// TIA Portal V15.1 export
// export: Created 2024-06-21T08:41:24.8000598Z, ExportSetting WithDefaults, DisplayName Totally Integrated Automation Portal, DisplayVersion V15.1 Update 5, DisplayName TIA Portal Openness, DisplayVersion V15.1 Update 5, DisplayName SINAMICS Startdrive Advanced, DisplayVersion V15.1, DisplayName G130, G150, S120, S150, SINAMICS MV, S210, DisplayVersion V15.1, DisplayName G110M, G120, G120C, G120D, G120P, DisplayVersion V15.1, DisplayName STEP 7 Professional, DisplayVersion V15.1 Update 5, DisplayName STEP 7 Safety, DisplayVersion V15.1, DisplayName WinCC Professional, DisplayVersion V15.1 Update 5, DisplayName SIMATIC Visualization Architect, DisplayVersion V15.1
FUNCTION "209230ZM01DataHandling" : Void   // FC404, FBD
TITLE = 209230ZM01 Data Handling
{ S7_Optimized_Access := 'FALSE' }
AUTHOR : VCC
VERSION : 0.1
// stored: AutoNumber false, IsIECCheckEnabled false, SetENOAutomatically False, UDAEnableTagReadback false
   VAR_OUTPUT
      O_AlarmA : Bool;   // Alarm A
      O_AlarmB : Bool;   // Alarm B
      O_AlarmC : Bool;   // Alarm C
      O_AlarmD : Bool;   // Alarm D
      O_AlarmABCondition : Bool;   // Alarm AB Condition
      H_IAnim : Word;   // Icon Animation
   END_VAR
BEGIN

REGION Network 1: **** 4.6 - Machine status - Indications **** Icon animation
   // Icon animation
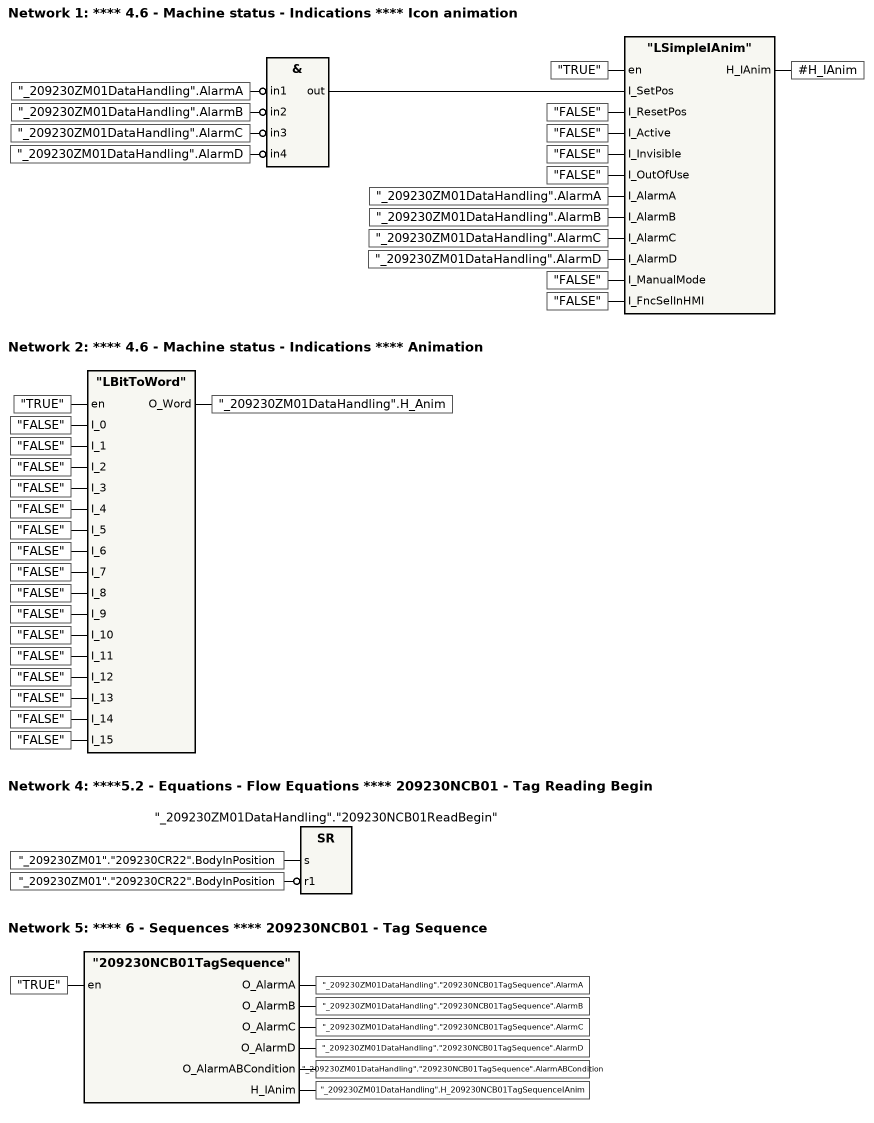
   IF "TRUE" THEN
       "LSimpleIAnim"(I_SetPos := NOT "_209230ZM01DataHandling".AlarmA AND NOT "_209230ZM01DataHandling".AlarmB AND NOT "_209230ZM01DataHandling".AlarmC AND NOT "_209230ZM01DataHandling".AlarmD,
                      I_ResetPos := "FALSE",
                      I_Active := "FALSE",
                      I_Invisible := "FALSE",
                      I_OutOfUse := "FALSE",
                      I_AlarmA := "_209230ZM01DataHandling".AlarmA,
                      I_AlarmB := "_209230ZM01DataHandling".AlarmB,
                      I_AlarmC := "_209230ZM01DataHandling".AlarmC,
                      I_AlarmD := "_209230ZM01DataHandling".AlarmD,
                      I_ManualMode := "FALSE",
                      I_FncSelInHMI := "FALSE",
                      H_IAnim => #H_IAnim);
   END_IF;
END_REGION

REGION Network 2: **** 4.6 - Machine status - Indications **** Animation
   // Animation
   IF "TRUE" THEN
       "LBitToWord"(I_0 := "FALSE",
                    I_1 := "FALSE",
                    I_2 := "FALSE",
                    I_3 := "FALSE",
                    I_4 := "FALSE",
                    I_5 := "FALSE",
                    I_6 := "FALSE",
                    I_7 := "FALSE",
                    I_8 := "FALSE",
                    I_9 := "FALSE",
                    I_10 := "FALSE",
                    I_11 := "FALSE",
                    I_12 := "FALSE",
                    I_13 := "FALSE",
                    I_14 := "FALSE",
                    I_15 := "FALSE",
                    O_Word => "_209230ZM01DataHandling".H_Anim);
   END_IF;
END_REGION

NETWORK
TITLE = **** 4.6 - Machine Status - Indications **** Animation DB number
// DB number
      OPN   "_209230ZM01DataHandling";
      L     DBNO;
      T     "_209230ZM01DataHandling".H_DBnr;

REGION Network 4: ****5.2 - Equations - Flow Equations **** 209230NCB01 - Tag Reading Begin
   // Singal to start the reading of the Tag
   IF "_209230ZM01"."209230CR22".BodyInPosition THEN
       "_209230ZM01DataHandling"."209230NCB01ReadBegin" := TRUE;   // SR flip-flop
   END_IF;
   IF NOT "_209230ZM01"."209230CR22".BodyInPosition THEN
       "_209230ZM01DataHandling"."209230NCB01ReadBegin" := FALSE;
   END_IF;
END_REGION

REGION Network 5: **** 6 - Sequences **** 209230NCB01 - Tag Sequence
   // Tag Sequence
   IF "TRUE" THEN
       "209230NCB01TagSequence"(O_AlarmA => "_209230ZM01DataHandling"."209230NCB01TagSequence".AlarmA,
                               O_AlarmB => "_209230ZM01DataHandling"."209230NCB01TagSequence".AlarmB,
                               O_AlarmC => "_209230ZM01DataHandling"."209230NCB01TagSequence".AlarmC,
                               O_AlarmD => "_209230ZM01DataHandling"."209230NCB01TagSequence".AlarmD,
                               O_AlarmABCondition => "_209230ZM01DataHandling"."209230NCB01TagSequence".AlarmABCondition,
                               H_IAnim => "_209230ZM01DataHandling".H_209230NCB01TagSequenceIAnim);
   END_IF;
END_REGION

REGION Network 6: **** 7.1 - Submodule - Non Machine **** 209230NCB01 - VIDS Master
   // VIDS Master Module
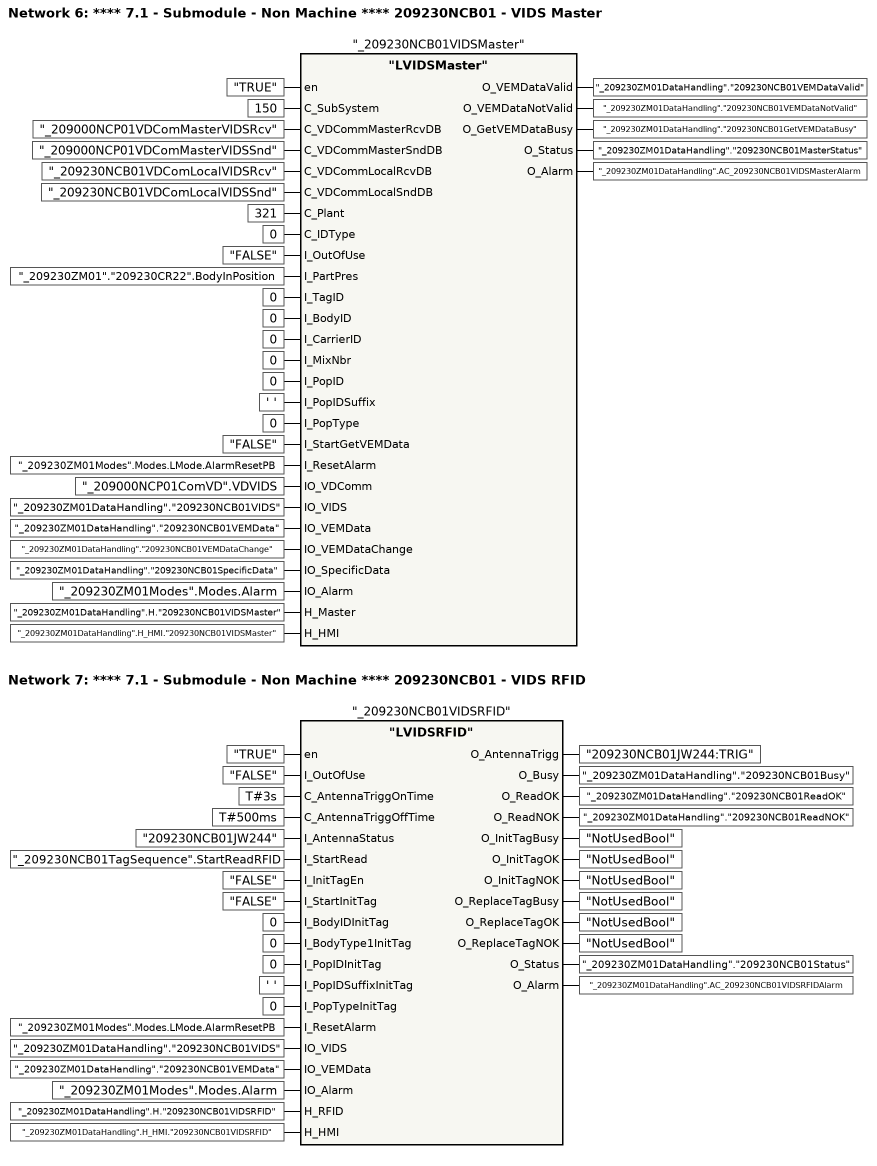
   IF "TRUE" THEN
       "_209230NCB01VIDSMaster"(C_SubSystem := 150,   // "LVIDSMaster"
                               C_VDCommMasterRcvDB := "_209000NCP01VDComMasterVIDSRcv",
                               C_VDCommMasterSndDB := "_209000NCP01VDComMasterVIDSSnd",
                               C_VDCommLocalRcvDB := "_209230NCB01VDComLocalVIDSRcv",
                               C_VDCommLocalSndDB := "_209230NCB01VDComLocalVIDSSnd",
                               C_Plant := 321,
                               C_IDType := 0,
                               I_OutOfUse := "FALSE",
                               I_PartPres := "_209230ZM01"."209230CR22".BodyInPosition,
                               I_TagID := 0,
                               I_BodyID := 0,
                               I_CarrierID := 0,
                               I_MixNbr := 0,
                               I_PopID := 0,
                               I_PopIDSuffix := ' ',
                               I_PopType := 0,
                               I_StartGetVEMData := "FALSE",
                               I_ResetAlarm := "_209230ZM01Modes".Modes.LMode.AlarmResetPB,
                               IO_VDComm := "_209000NCP01ComVD".VDVIDS,
                               IO_VIDS := "_209230ZM01DataHandling"."209230NCB01VIDS",
                               IO_VEMData := "_209230ZM01DataHandling"."209230NCB01VEMData",
                               IO_VEMDataChange := "_209230ZM01DataHandling"."209230NCB01VEMDataChange",
                               IO_SpecificData := "_209230ZM01DataHandling"."209230NCB01SpecificData",
                               IO_Alarm := "_209230ZM01Modes".Modes.Alarm,
                               H_Master := "_209230ZM01DataHandling".H."209230NCB01VIDSMaster",
                               H_HMI := "_209230ZM01DataHandling".H_HMI."209230NCB01VIDSMaster",
                               O_VEMDataValid => "_209230ZM01DataHandling"."209230NCB01VEMDataValid",
                               O_VEMDataNotValid => "_209230ZM01DataHandling"."209230NCB01VEMDataNotValid",
                               O_GetVEMDataBusy => "_209230ZM01DataHandling"."209230NCB01GetVEMDataBusy",
                               O_Status => "_209230ZM01DataHandling"."209230NCB01MasterStatus",
                               O_Alarm => "_209230ZM01DataHandling".AC_209230NCB01VIDSMasterAlarm);
   END_IF;
END_REGION

REGION Network 7: **** 7.1 - Submodule - Non Machine **** 209230NCB01 - VIDS RFID
   // VIDS RFID Module
   IF "TRUE" THEN
       "_209230NCB01VIDSRFID"(I_OutOfUse := "FALSE",   // "LVIDSRFID"
                              C_AntennaTriggOnTime := T#3s,
                              C_AntennaTriggOffTime := T#500ms,
                              I_AntennaStatus := "209230NCB01JW244",
                              I_StartRead := "_209230NCB01TagSequence".StartReadRFID,
                              I_InitTagEn := "FALSE",
                              I_StartInitTag := "FALSE",
                              I_BodyIDInitTag := 0,
                              I_BodyType1InitTag := 0,
                              I_PopIDInitTag := 0,
                              I_PopIDSuffixInitTag := ' ',
                              I_PopTypeInitTag := 0,
                              I_ResetAlarm := "_209230ZM01Modes".Modes.LMode.AlarmResetPB,
                              IO_VIDS := "_209230ZM01DataHandling"."209230NCB01VIDS",
                              IO_VEMData := "_209230ZM01DataHandling"."209230NCB01VEMData",
                              IO_Alarm := "_209230ZM01Modes".Modes.Alarm,
                              H_RFID := "_209230ZM01DataHandling".H."209230NCB01VIDSRFID",
                              H_HMI := "_209230ZM01DataHandling".H_HMI."209230NCB01VIDSRFID",
                              O_AntennaTrigg => "209230NCB01JW244:TRIG",
                              O_Busy => "_209230ZM01DataHandling"."209230NCB01Busy",
                              O_ReadOK => "_209230ZM01DataHandling"."209230NCB01ReadOK",
                              O_ReadNOK => "_209230ZM01DataHandling"."209230NCB01ReadNOK",
                              O_InitTagBusy => "NotUsedBool",
                              O_InitTagOK => "NotUsedBool",
                              O_InitTagNOK => "NotUsedBool",
                              O_ReplaceTagBusy => "NotUsedBool",
                              O_ReplaceTagOK => "NotUsedBool",
                              O_ReplaceTagNOK => "NotUsedBool",
                              O_Status => "_209230ZM01DataHandling"."209230NCB01Status",
                              O_Alarm => "_209230ZM01DataHandling".AC_209230NCB01VIDSRFIDAlarm);
   END_IF;
END_REGION

REGION Network 8: **** 7.1 - Submodule - Non Machine ****209230NCB01 - VIDS Tracking
   // VIDS Tracking Module
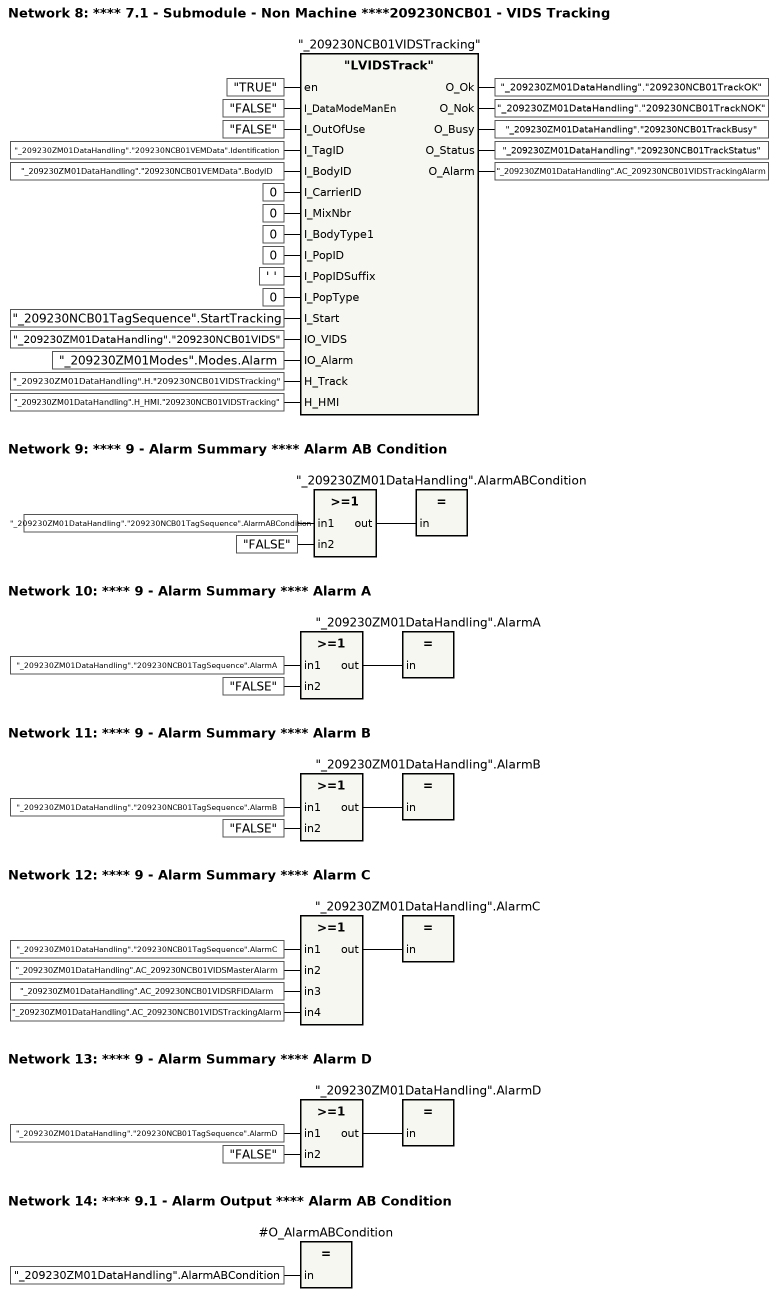
   IF "TRUE" THEN
       "_209230NCB01VIDSTracking"(I_DataModeManEn := "FALSE",   // "LVIDSTrack"
                               I_OutOfUse := "FALSE",
                               I_TagID := "_209230ZM01DataHandling"."209230NCB01VEMData".Identification,
                               I_BodyID := "_209230ZM01DataHandling"."209230NCB01VEMData".BodyID,
                               I_CarrierID := 0,
                               I_MixNbr := 0,
                               I_BodyType1 := 0,
                               I_PopID := 0,
                               I_PopIDSuffix := ' ',
                               I_PopType := 0,
                               I_Start := "_209230NCB01TagSequence".StartTracking,
                               IO_VIDS := "_209230ZM01DataHandling"."209230NCB01VIDS",
                               IO_Alarm := "_209230ZM01Modes".Modes.Alarm,
                               H_Track := "_209230ZM01DataHandling".H."209230NCB01VIDSTracking",
                               H_HMI := "_209230ZM01DataHandling".H_HMI."209230NCB01VIDSTracking",
                               O_Ok => "_209230ZM01DataHandling"."209230NCB01TrackOK",
                               O_Nok => "_209230ZM01DataHandling"."209230NCB01TrackNOK",
                               O_Busy => "_209230ZM01DataHandling"."209230NCB01TrackBusy",
                               O_Status => "_209230ZM01DataHandling"."209230NCB01TrackStatus",
                               O_Alarm => "_209230ZM01DataHandling".AC_209230NCB01VIDSTrackingAlarm);
   END_IF;
END_REGION

REGION Network 9: **** 9 - Alarm Summary **** Alarm AB Condition
   // Alarm AB Condition
   "_209230ZM01DataHandling".AlarmABCondition := "_209230ZM01DataHandling"."209230NCB01TagSequence".AlarmABCondition OR "FALSE";
END_REGION

REGION Network 10: **** 9 - Alarm Summary **** Alarm A
   // Alarm A
   "_209230ZM01DataHandling".AlarmA := "_209230ZM01DataHandling"."209230NCB01TagSequence".AlarmA OR "FALSE";
END_REGION

REGION Network 11: **** 9 - Alarm Summary **** Alarm B
   // Alarm B
   "_209230ZM01DataHandling".AlarmB := "_209230ZM01DataHandling"."209230NCB01TagSequence".AlarmB OR "FALSE";
END_REGION

REGION Network 12: **** 9 - Alarm Summary **** Alarm C
   // Alarm C
   "_209230ZM01DataHandling".AlarmC := "_209230ZM01DataHandling"."209230NCB01TagSequence".AlarmC OR "_209230ZM01DataHandling".AC_209230NCB01VIDSMasterAlarm OR "_209230ZM01DataHandling".AC_209230NCB01VIDSRFIDAlarm OR "_209230ZM01DataHandling".AC_209230NCB01VIDSTrackingAlarm;
END_REGION

REGION Network 13: **** 9 - Alarm Summary **** Alarm D
   // Alarm D
   "_209230ZM01DataHandling".AlarmD := "_209230ZM01DataHandling"."209230NCB01TagSequence".AlarmD OR "FALSE";
END_REGION

REGION Network 14: **** 9.1 - Alarm Output **** Alarm AB Condition
   // Alarm AB Condition
   #O_AlarmABCondition := "_209230ZM01DataHandling".AlarmABCondition;
END_REGION

REGION Network 15: **** 9.1 - Alarm Output **** Alarm A
   // Alarm A
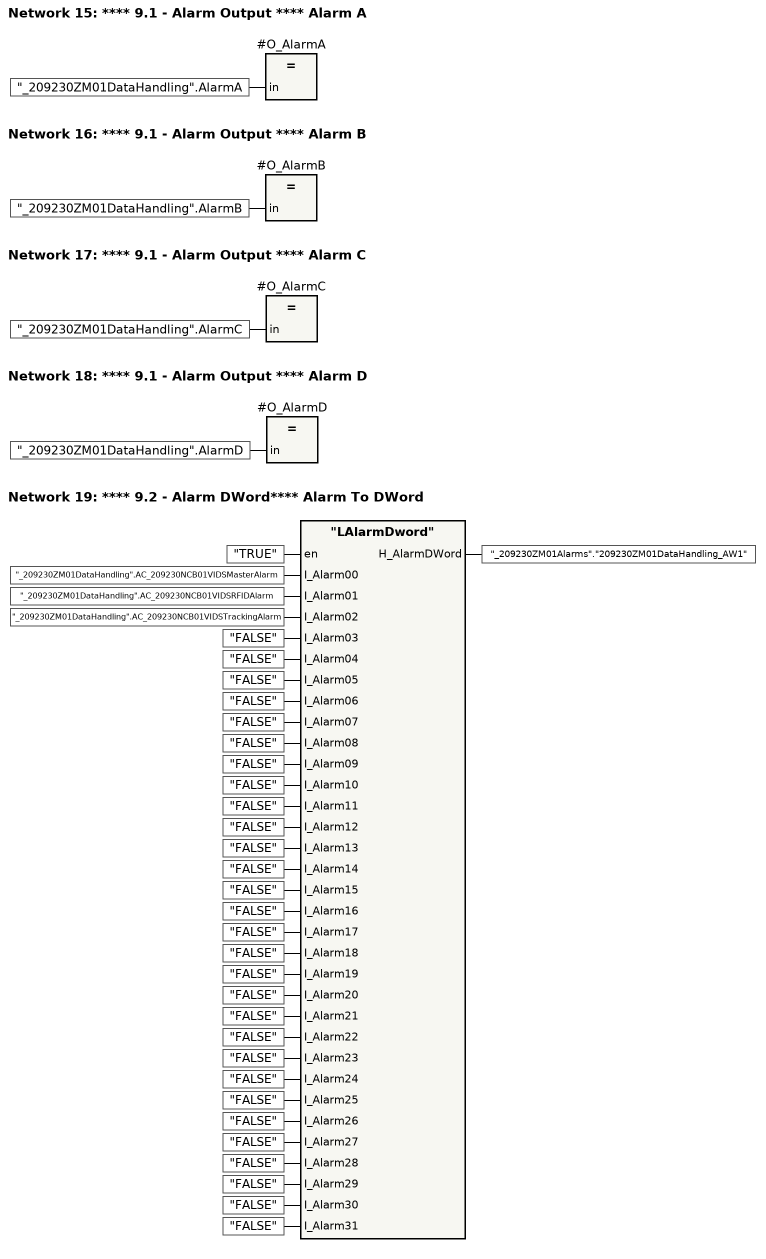
   #O_AlarmA := "_209230ZM01DataHandling".AlarmA;
END_REGION

REGION Network 16: **** 9.1 - Alarm Output **** Alarm B
   // Alarm B
   #O_AlarmB := "_209230ZM01DataHandling".AlarmB;
END_REGION

REGION Network 17: **** 9.1 - Alarm Output **** Alarm C
   // Alarm C
   #O_AlarmC := "_209230ZM01DataHandling".AlarmC;
END_REGION

REGION Network 18: **** 9.1 - Alarm Output **** Alarm D
   // Alarm D
   #O_AlarmD := "_209230ZM01DataHandling".AlarmD;
END_REGION

REGION Network 19: **** 9.2 - Alarm DWord**** Alarm To DWord
   // Alarm Word
   IF "TRUE" THEN
       "LAlarmDword"(I_Alarm00 := "_209230ZM01DataHandling".AC_209230NCB01VIDSMasterAlarm,
                     I_Alarm01 := "_209230ZM01DataHandling".AC_209230NCB01VIDSRFIDAlarm,
                     I_Alarm02 := "_209230ZM01DataHandling".AC_209230NCB01VIDSTrackingAlarm,
                     I_Alarm03 := "FALSE",
                     I_Alarm04 := "FALSE",
                     I_Alarm05 := "FALSE",
                     I_Alarm06 := "FALSE",
                     I_Alarm07 := "FALSE",
                     I_Alarm08 := "FALSE",
                     I_Alarm09 := "FALSE",
                     I_Alarm10 := "FALSE",
                     I_Alarm11 := "FALSE",
                     I_Alarm12 := "FALSE",
                     I_Alarm13 := "FALSE",
                     I_Alarm14 := "FALSE",
                     I_Alarm15 := "FALSE",
                     I_Alarm16 := "FALSE",
                     I_Alarm17 := "FALSE",
                     I_Alarm18 := "FALSE",
                     I_Alarm19 := "FALSE",
                     I_Alarm20 := "FALSE",
                     I_Alarm21 := "FALSE",
                     I_Alarm22 := "FALSE",
                     I_Alarm23 := "FALSE",
                     I_Alarm24 := "FALSE",
                     I_Alarm25 := "FALSE",
                     I_Alarm26 := "FALSE",
                     I_Alarm27 := "FALSE",
                     I_Alarm28 := "FALSE",
                     I_Alarm29 := "FALSE",
                     I_Alarm30 := "FALSE",
                     I_Alarm31 := "FALSE",
                     H_AlarmDWord => "_209230ZM01Alarms"."209230ZM01DataHandling_AW1");
   END_IF;
END_REGION
END_FUNCTION
